FUNCTION_BLOCK valve_digital
VAR_INPUT
	//Open Feedback from Valve
	open_feedback : BOOL; 
	//Closed Feedback from Valve
	closed_feedback : BOOL;
	//Open Request from PLC Program
	open_request : BOOL;
	//Triggered from alarm ladder
	fault : BOOL;
END_VAR
VAR_OUTPUT
	//Tells the valve to open when true, close when False
	open_command : BOOL;
	// Valve status, 0=Closed, 1=Open, 2=Faulted
	status: INT;
END_VAR
VAR	
END_VAR
VAR // added by the converter: edge detectors and wires of the graphical bodies
    _w1, _w2, _w3 : BOOL;
END_VAR

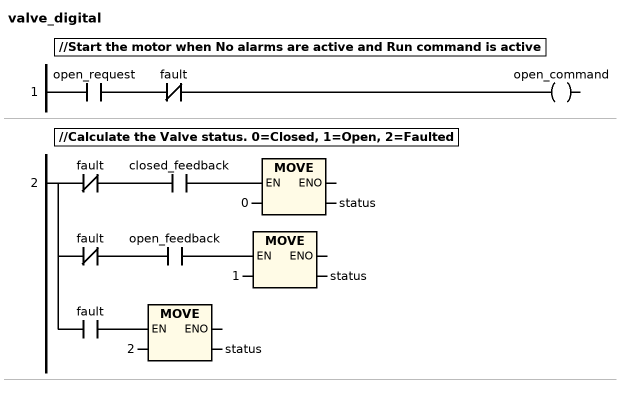
// NETWORK 1
// label: //Start the motor when No alarms are active and Run command is active
open_command := open_request AND NOT fault;

// NETWORK 2
// label: //Calculate the Valve status. 0=Closed, 1=Open, 2=Faulted
_w1 := NOT fault AND closed_feedback;
IF _w1 THEN status := 0; END_IF
_w2 := NOT fault AND open_feedback;
IF _w2 THEN status := 1; END_IF
_w3 := fault;
IF _w3 THEN status := 2; END_IF

END_FUNCTION_BLOCK

(* stored: Version 1.1.0.1, ProductVersion 3.1.4024.12
   POU valve_digital: Id {98e771d8-3fe1-4057-aa61-fd7121110cde}, SpecialFunc None *)
